// TIA Portal project "scl_1buton_2motor_tetikleme" (V18)

(* hardware
DEVICE "S7-1200 station_1"  S7-1200 Station
   slot 0: "Rack_0"  S7-1200 Rack  Rack  V1.0
   slot 1: "PLC_1"  CPU 1214C DC/DC/DC  6ES7 214-1AG40-0XB0  V4.6
*)

// ===== PLC "PLC_1"  CPU 1214C DC/DC/DC =====

VAR_GLOBAL   // PLC tag table "Default tag table"
   "STOP" AT %I0.0 : Bool;
   "START" AT %I0.1 : Bool;
   "MOTOR_1" AT %Q0.0 : Bool;
   "MOTOR_2" AT %Q0.1 : Bool;
   "pozitif kenar tetikleme merker" AT %M0.0 : Bool;
   "pozitif yardımcı kenar tetikleme merker" AT %M0.1 : Bool;
   "negatif kenar tetikleme merker" AT %M0.2 : Bool;
   "negatif yardımcı kenar tetikleme merker" AT %M0.3 : Bool;
END_VAR

FUNCTION "Block_1" : Void   // FC1, SCL
{ S7_Optimized_Access := 'TRUE' }
VERSION : 0.1
BEGIN
   "pozitif kenar tetikleme merker" := "START" AND NOT "pozitif yardımcı kenar tetikleme merker";
   "pozitif yardımcı kenar tetikleme merker" := "START";

   "negatif kenar tetikleme merker" := "negatif yardımcı kenar tetikleme merker" AND NOT "START";
   "negatif yardımcı kenar tetikleme merker" := "START";

   IF "pozitif kenar tetikleme merker"=1 THEN
       "MOTOR_1" := 1;
       "MOTOR_2" := 1;
   END_IF;

   IF "negatif kenar tetikleme merker"=1 THEN
       "MOTOR_1" := 0;
       "MOTOR_2" := 1;
   END_IF;

   IF "STOP" = 1 THEN
       "MOTOR_1" := 0;
       "MOTOR_2" := 0;
   END_IF;
END_FUNCTION

ORGANIZATION_BLOCK "Main"   // OB1, LAD, ProgramCycle
TITLE = "Main Program Sweep (Cycle)"
{ S7_Optimized_Access := 'TRUE' }
VERSION : 0.1
   VAR_INPUT
      Initial_Call : Bool;   // Initial call of this OB
      Remanence : Bool;   // =True, if remanent data are available
   END_VAR
BEGIN
END_ORGANIZATION_BLOCK